// LS Electric XG5000 project: traffic lights
// PLC NewPLC

PROGRAM NewProgram (task: Scan Program)

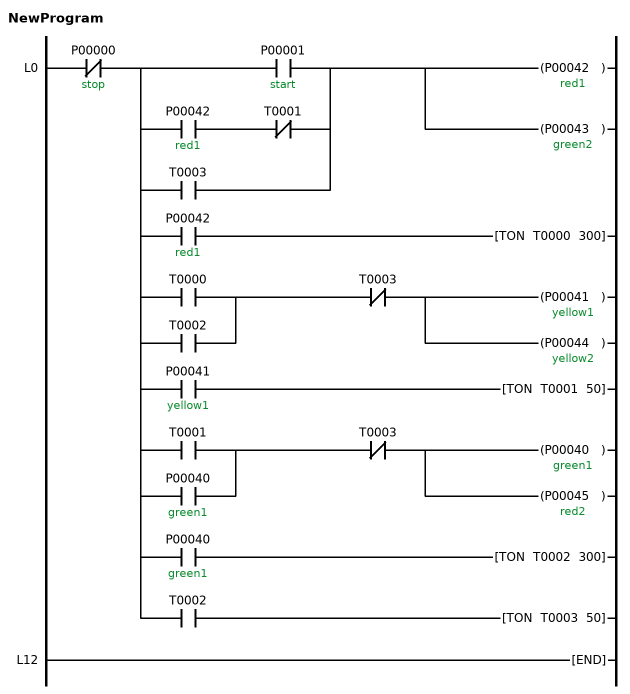
; L0
LOAD NOT  P00000	// stop
MPUSH
LOAD      P00001	// start
LOAD      P00042	// red1
AND NOT   T0001
OR LOAD
OR        T0003
AND LOAD
OUT       P00042	// red1
OUT       P00043	// green2
MLOAD
AND       P00042	// red1
TON       T0000 300
MLOAD
LOAD      T0000
OR        T0002
AND LOAD
AND NOT   T0003
OUT       P00041	// yellow1
OUT       P00044	// yellow2
MLOAD
AND       P00041	// yellow1
TON       T0001 50
MLOAD
LOAD      T0001
OR        P00040	// green1
AND LOAD
AND NOT   T0003
OUT       P00040	// green1
OUT       P00045	// red2
MLOAD
AND       P00040	// green1
TON       T0002 300
MPOP
AND       T0002
TON       T0003 50
; L12
END